FUNCTION_BLOCK FB_UML_SC_Composite
VAR	
	bInitFinished			: BOOL;
	bUseXmlFormat			: BOOL;
	bAllInfoCopiedToFile	: BOOL;
	bSendToMasterFinished	: BOOL;
	bSendToClientFinished	: BOOL;
END_VAR

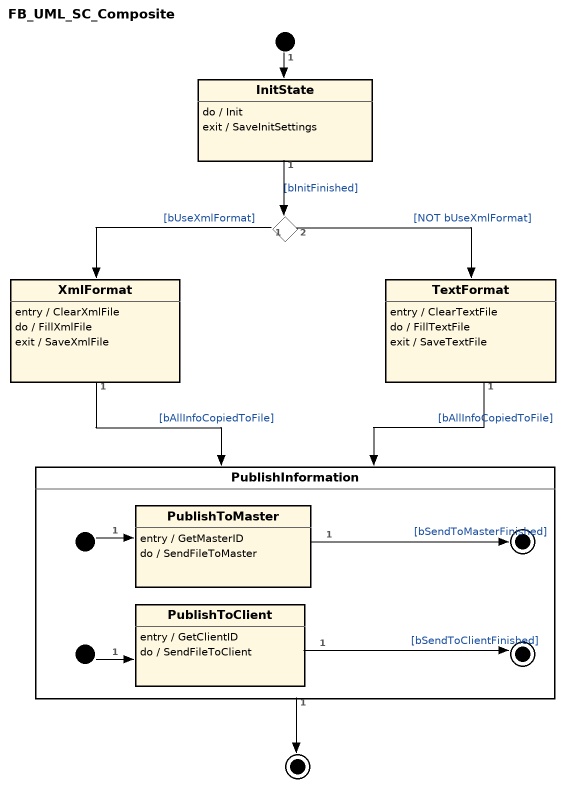
STATECHART FB_UML_SC_Composite  // abortable
    START StartState1
    STATE InitState
        do / Init
        exit / SaveInitSettings
    CHOICE ChoiceElement1
    STATE XmlFormat
        entry / ClearXmlFile
        do / FillXmlFile
        exit / SaveXmlFile
    STATE TextFormat
        entry / ClearTextFile
        do / FillTextFile
        exit / SaveTextFile
    COMPOSITE STATE PublishInformation
        REGION Region1 // priority 1
        START StartState3
        STATE PublishToClient
            entry / GetClientID
            do / SendFileToClient
        END EndState3
        StartState3 -> PublishToClient  // priority 1, on completion
        PublishToClient -> EndState3 [bSendToClientFinished] // priority 1
        REGION Region0 // priority 2
        START StartState2
        STATE PublishToMaster
            entry / GetMasterID
            do / SendFileToMaster
        END EndState2
        StartState2 -> PublishToMaster  // priority 1, on completion
        PublishToMaster -> EndState2 [bSendToMasterFinished] // priority 1
    END_STATE
    END EndState1
    StartState1 -> InitState  // priority 1, on completion
    InitState -> ChoiceElement1 [bInitFinished] // priority 1
    ChoiceElement1 -> XmlFormat [bUseXmlFormat] // priority 1
    ChoiceElement1 -> TextFormat [NOT bUseXmlFormat] // priority 2
    XmlFormat -> PublishInformation [bAllInfoCopiedToFile] // priority 1
    TextFormat -> PublishInformation [bAllInfoCopiedToFile] // priority 1
    PublishInformation -> EndState1  // priority 1, on completion
END_STATECHART

ACTION ClearTextFile:
nCounterClearText := nCounterClearText + 1;
END_ACTION

ACTION ClearXmlFile:
nCounterClearXml := nCounterClearXml + 1;
END_ACTION

ACTION FillTextFile:
nCounterFillText := nCounterFillText + 1;
END_ACTION

ACTION FillXmlFile:
nCounterFillXml := nCounterFillXml + 1;
END_ACTION

ACTION GetClientID:
nCounterGetClientID := nCounterGetClientID + 1;

IF nCounterGetClientID = 1 AND nCounterGetMasterID = 0 THEN
	bClientFirst := TRUE;
END_IF
END_ACTION

ACTION GetMasterID:
nCounterGetMasterID := nCounterGetMasterID + 1;

IF nCounterGetClientID = 0 AND nCounterGetMasterID = 1 THEN
	bMasterFirst := TRUE;
END_IF
END_ACTION

ACTION Init:
nCounterInit := nCounterInit + 1;
END_ACTION

ACTION SaveInitSettings:
nCounterSaveInitSettings := nCounterSaveInitSettings + 1;

bInitFinished 			:= FALSE;
bAllInfoCopiedToFile 	:= FALSE;
bSendToClientFinished 	:= FALSE;
bSendToMasterFinished	:= FALSE;
END_ACTION

ACTION SaveTextFile:
nCounterSaveText := nCounterSaveText + 1;
END_ACTION

ACTION SaveXmlFile:
nCounterSaveXml := nCounterSaveXml + 1;
END_ACTION

ACTION SendFileToClient:
nCounterSendToClient := nCounterSendToClient + 1;
END_ACTION

ACTION SendFileToMaster:
nCounterSendToMaster := nCounterSendToMaster + 1;
END_ACTION

END_FUNCTION_BLOCK

(* stored: Version 1.1.0.1, ProductVersion 3.1.4024.11
   POU FB_UML_SC_Composite: Id {94bc9ba2-99d4-44d6-a994-09cf55f5519b}, SpecialFunc None
   Action ClearTextFile: Id {0bb73ff2-7d6d-417f-9c12-5132b03a4a13}
   Action ClearXmlFile: Id {d0aa2933-34a3-48a1-aee6-eb675a6fe610}
   Action FillTextFile: Id {8a647094-38df-418e-9700-18e100a5485e}
   Action FillXmlFile: Id {b2718471-98be-4693-87c2-538162020aec}
   Action GetClientID: Id {a93eeae2-d85f-4f20-943f-0afd788e65ee}
   Action GetMasterID: Id {c3ed8ce0-dda3-4a83-9da9-a0dbf863c4dc}
   Action Init: Id {90a717ec-c5e9-4f4f-9dc6-eaf3c84211c2}
   Action SaveInitSettings: Id {7be3acb2-a8f9-4548-a342-1b987d1d3829}
   Action SaveTextFile: Id {4181e14c-23b8-49c9-8fe1-51425b6bd4f6}
   Action SaveXmlFile: Id {39d485de-ff2b-4f11-8ae4-b1b9701fa0c8}
   Action SendFileToClient: Id {24f8047c-7cc5-4260-a8fe-c1c08e37fe8f}
   Action SendFileToMaster: Id {a64eb469-9952-480a-9ea3-33cc4500d480} *)
